Universal Robots PolyScope program: CORAL_QR_l3.urp

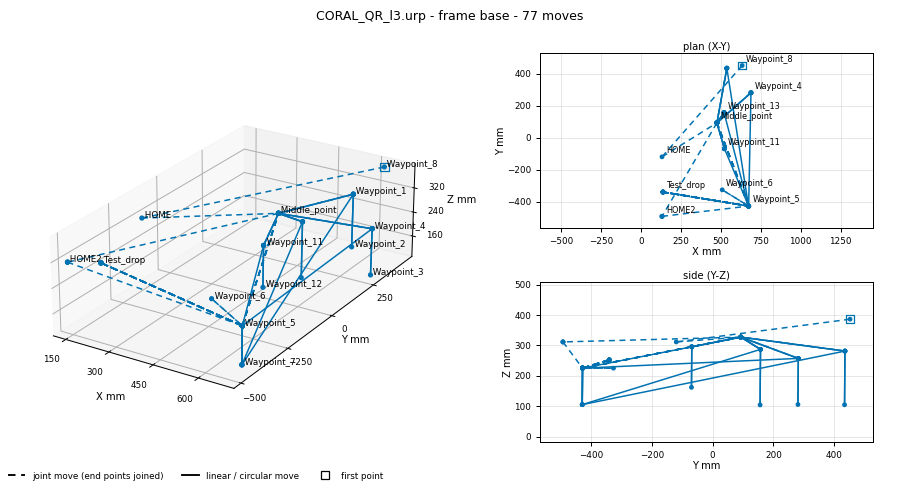
[picture p0: tool path of CORAL_QR_l3.urp in frame base, 77 of 90 moves have a stored position in this frame; points joined in program order, loops and branches not executed]
Program CORAL_QR_l3 (installation=CORAL_installation directory=/programs/usbdisk_0 createdIn=5.13.0 lastSavedIn=5.13.0 robotSerialNumber=20215502618)
Calibrated DH parameters: a=[0.000207, -0.251803, -0.392414, 0.000115, 0.000037, 0]; d=[0.162602, -473.711772, 472.954062, 0.891293, 0.099607, 0.099704]; alpha=[1.571111, -0.000723, 0.005186, 1.570255, -1.569363, 0]; deltaTheta=[0, 0.936857, 5.33632, 0.010013, 0, 0]
InitVariablesNode
Robot Program (runOnlyOnce=false)
  pos_3 := p[0.22031,-0.00393,-0.14981,0.011,-0.001,-1.563]
  pos_4 := p[0.58548,-0.15484,-0.12328,0.011,-0.001,-1.594]
  pos_5 := p[0.38723,-0.17108,-0.15474,0.011,-0.001,-1.594]
  distance := p[0,-0.1,0,0,0,0]
  cont_1 := 1
  cont_2 := 1
  cont_3 := 2
  cont_4 := 2
  cont_5 := 2
  cont_6 := 1
  cont_7 := 1
  no_object := 0
  URCap Gripper Activate (Robotiq_Grippers, Robotiq Inc.) dataModel(ResetAndActivateKey=true)
  URCap External Control (External Control, FZI Research Center for Information Technology)
  MoveL speed 250 mm/s, acceleration 1200 mm/s^2 (useActiveTCP=true) feature=Base
    Waypoint Waypoint_8: TCP in base x=634.227 y=451.95 z=386.422 mm, rx=-1.7963 ry=2.0874 rz=0.1446 rad; joints [201.008, -64.187, 54.919, -99.703, -76.956, 31.795] deg; TCP offset x=0 y=0 z=175.5 mm, rx=0 ry=0 rz=0 rad
  URCap Find Visual Offset (Robotiq_Wrist_Camera, Robotiq Inc.) dataModel(tagModel=[{"_featureName":"CORAL","_automaticMoveEnabled":false,"_ignoreSnapshotPositionEnabled":true,"_skipCloseSnapshotPositionEnabled":false}]); state(isChildrenLocked=true)
    URCap If tag found (Robotiq_Wrist_Camera, Robotiq Inc.)
      URCap Apply Visual Offset (Robotiq_Wrist_Camera, Robotiq Inc.) dataModel(tagModel=[{"_featureName":"CORAL","_appliedEverywhere":false}])
        'Tag found'
        URCap Gripper (Robotiq_Grippers, Robotiq Inc.) dataModel(position=0.0, force=0.0, speed=0.0, positionInDouble=0.0, forceInDouble=0.0, speedInDouble=0.0, slaveIds=[9], blocking=true)
        Loop Forever
          URCap Gripper (Robotiq_Grippers, Robotiq Inc.) dataModel(position=0.0, force=0.0, speed=0.0, positionInDouble=0.0, forceInDouble=0.0, speedInDouble=0.0, slaveIds=[9], blocking=true)
          MoveJ speed 60 deg/s, acceleration 80 deg/s^2 (useActiveTCP=true) feature=Base
            Waypoint HOME: TCP in base x=132.452 y=-119.516 z=311.713 mm, rx=0.0014 ry=-3.1367 rz=0.0022 rad; joints [90.048, -142.3, 117.416, -65.113, -89.996, -0.059] deg
          Wait Condition expression=binary_list_to_integer([digital_in[3],digital_in[4],digital_in[5],digital_in[6],digital_in[7]])==0
          Wait Sleep waitTime=0.25
          Wait Condition expression=binary_list_to_integer([digital_in[3],digital_in[4],digital_in[5],digital_in[6],digital_in[7]])≠0
          Wait Sleep waitTime=0.25
          Script: bit=[digital_in[3],digital_in[4],digital_in[5],digital_in[6],digital_in[7]]
          If binary_list_to_integer(bit)==20
            Wait Condition expression=binary_list_to_integer([digital_in[3],digital_in[4],digital_in[5],digital_in[6],digital_in[7]])==0
            Wait Sleep waitTime=0.25
            Wait Condition expression=binary_list_to_integer([digital_in[3],digital_in[4],digital_in[5],digital_in[6],digital_in[7]])≠0
            Wait Sleep waitTime=0.25
            Script: bit=[digital_in[3],digital_in[4],digital_in[5],digital_in[6],digital_in[7]]
            object := binary_list_to_integer(bit)
            Switch expression=object
              Case (caseValue=11)
                If cont_1≥1
                  MoveJ speed 60 deg/s, acceleration 80 deg/s^2 (useActiveTCP=false) tcp=Robotiq_2F85; feature=Base
                    Waypoint Middle_point: TCP in base x=476.066 y=92.919 z=327.558 mm, rx=-2.1236 ry=2.3147 rz=-0.0001 rad; joints [175.026, -93.413, 90.975, -87.495, -89.706, -0.002] deg
                  MoveL speed 250 mm/s, acceleration 1200 mm/s^2 (useActiveTCP=false) tcp=Robotiq_2F85; feature=CORAL
                    Waypoint Waypoint_1: TCP in base x=538.261 y=435.272 z=281.637 mm, rx=-2.2567 ry=2.1855 rz=-0.0001 rad; joints [207.833, -63.818, 61.827, -87.934, -89.728, 26.021] deg; feature pose in base x=487.974 y=527.462 z=106.955 mm, rx=2.2289 ry=-2.2003 rz=0.002 rad
                    Waypoint Waypoint_2: TCP in base x=537.232 y=433.915 z=104.968 mm, rx=-2.2568 ry=2.1854 rz=-0.0001 rad; joints [207.75, -59.619, 81.826, -112.131, -89.748, 26.056] deg
                    URCap Gripper (Robotiq_Grippers, Robotiq Inc.) dataModel(position=100.0, force=0.0, speed=50.0, positionInDouble=100.0, forceInDouble=0.0, speedInDouble=50.0, slaveIds=[9], blocking=true)
                    Waypoint Waypoint_1: TCP in base x=538.261 y=435.272 z=281.637 mm, rx=-2.2567 ry=2.1855 rz=-0.0001 rad; joints [207.833, -63.818, 61.827, -87.934, -89.728, 26.021] deg
                  cont_1 := cont_1-1
                  no_object := 0
                Else 
                  no_object := 1
                  Popup Message (haltProgram=false message=Out of stock! inputType=Text)
              Case (caseValue=12)
                If cont_2≥1
                  MoveJ speed 60 deg/s, acceleration 80 deg/s^2 (useActiveTCP=false) tcp=Robotiq_2F85; feature=Base
                    Waypoint Middle_point: TCP in base x=476.066 y=92.919 z=327.558 mm, rx=-2.1236 ry=2.3147 rz=-0.0001 rad; joints [175.026, -93.413, 90.975, -87.495, -89.706, -0.002] deg
                  MoveL speed 250 mm/s, acceleration 1200 mm/s^2 (useActiveTCP=false) tcp=Robotiq_2F85; feature=CORAL
                    Waypoint Waypoint_4: TCP in base x=689.362 y=281.81 z=257.546 mm, rx=3.1339 ry=0.0106 rz=-0.0087 rad; joints [192.043, -55.015, 51.59, -86.091, -90.092, -78.333] deg; feature pose in base x=487.974 y=527.462 z=106.955 mm, rx=2.2289 ry=-2.2003 rz=0.002 rad
                    Waypoint Waypoint_3: TCP in base x=688.512 y=280.634 z=105.968 mm, rx=3.1339 ry=0.0105 rz=-0.0087 rad; joints [191.949, -52.35, 69.613, -106.779, -90.102, -78.321] deg
                    URCap Gripper (Robotiq_Grippers, Robotiq Inc.) dataModel(position=100.0, force=0.0, speed=50.0, positionInDouble=100.0, forceInDouble=0.0, speedInDouble=50.0, slaveIds=[9], blocking=true)
                    Waypoint Waypoint_4: TCP in base x=689.362 y=281.81 z=257.546 mm, rx=3.1339 ry=0.0106 rz=-0.0087 rad; joints [192.043, -55.015, 51.59, -86.091, -90.092, -78.333] deg
                  cont_2 := cont_2-1
                  no_object := 0
                Else 
                  no_object := 1
                  Popup Message (haltProgram=false message=Out of stock! inputType=Text)
              Case (caseValue=13)
                If cont_3≥1
                  MoveJ speed 60 deg/s, acceleration 80 deg/s^2 (useActiveTCP=false) tcp=Robotiq_2F85; feature=Base
                    Waypoint Middle_point: TCP in base x=476.066 y=92.919 z=327.558 mm, rx=-2.1236 ry=2.3147 rz=-0.0001 rad; joints [175.026, -93.413, 90.975, -87.495, -89.706, -0.002] deg
                  MoveL speed 250 mm/s, acceleration 1200 mm/s^2 (useActiveTCP=false) tcp=Robotiq_2F85; feature=CORAL
                    Waypoint Variable (Variable): variable=pos_3
                    MoveDirectionNode (selectedDirection=ZPlus toolParams=0.07, 1.2)
                      Until TOOL_CONTACT_DETECTION (allowActions=false retraction=0.02 decelerationAcceleration=3 decelerationAngularAcceleration=34.906585)
                      SuppressedNode
                        Until DISTANCE (allowActions=false deceleration=3 distanceNodeType=STOP) Distance=0.14904; motionParameters(blendRadius=0)
                    URCap Gripper (Robotiq_Grippers, Robotiq Inc.) dataModel(position=100.0, force=0.0, speed=50.0, positionInDouble=100.0, forceInDouble=0.0, speedInDouble=50.0, slaveIds=[9], blocking=true)
                    Waypoint Variable (Variable): variable=pos_3
                    pos_3 := pose_add(pos_3, distance)
                    cont_3 := cont_3-1
                    no_object := 0
                Else 
                  no_object := 1
                  Popup Message (haltProgram=false message=Out of stock! inputType=Text)
              Case (caseValue=14)
                If cont_4≥1
                  MoveJ speed 60 deg/s, acceleration 80 deg/s^2 (useActiveTCP=false) tcp=Robotiq_2F85; feature=Base
                    Waypoint Middle_point: TCP in base x=476.066 y=92.919 z=327.558 mm, rx=-2.1236 ry=2.3147 rz=-0.0001 rad; joints [175.026, -93.413, 90.975, -87.495, -89.706, -0.002] deg
                  MoveL speed 250 mm/s, acceleration 1200 mm/s^2 (useActiveTCP=false) tcp=Robotiq_2F85; feature=CORAL
                    Waypoint Variable (Variable): variable=pos_4
                    MoveDirectionNode (selectedDirection=ZPlus toolParams=0.07, 1.2)
                      Until TOOL_CONTACT_DETECTION (allowActions=false retraction=0.02 decelerationAcceleration=3 decelerationAngularAcceleration=34.906585)
                      SuppressedNode
                        Until DISTANCE (allowActions=false deceleration=3 distanceNodeType=STOP) Distance=0.13; motionParameters(blendRadius=0)
                    URCap Gripper (Robotiq_Grippers, Robotiq Inc.) dataModel(position=100.0, force=0.0, speed=50.0, positionInDouble=100.0, forceInDouble=0.0, speedInDouble=50.0, slaveIds=[9], blocking=true)
                    Waypoint Variable (Variable): variable=pos_4
                    pos_4 := pose_add(pos_4, distance)
                    cont_4 := cont_4-1
                    no_object := 0
                Else 
                  no_object := 1
                  Popup Message (haltProgram=false message=Out of stock! inputType=Text)
              Case (caseValue=15)
                If cont_5≥1
                  MoveJ speed 60 deg/s, acceleration 80 deg/s^2 (useActiveTCP=false) tcp=Robotiq_2F85; feature=Base
                    Waypoint Middle_point: TCP in base x=476.066 y=92.919 z=327.558 mm, rx=-2.1236 ry=2.3147 rz=-0.0001 rad; joints [175.026, -93.413, 90.975, -87.495, -89.706, -0.002] deg
                  MoveL speed 250 mm/s, acceleration 1200 mm/s^2 (useActiveTCP=false) tcp=Robotiq_2F85; feature=CORAL
                    Waypoint Variable (Variable): variable=pos_5
                    MoveDirectionNode (selectedDirection=ZPlus toolParams=0.07, 1.2)
                      Until TOOL_CONTACT_DETECTION (allowActions=false retraction=0.02 decelerationAcceleration=3 decelerationAngularAcceleration=34.906585)
                      SuppressedNode
                        Until DISTANCE (allowActions=false deceleration=3 distanceNodeType=STOP) Distance=0.1485; motionParameters(blendRadius=0)
                    URCap Gripper (Robotiq_Grippers, Robotiq Inc.) dataModel(position=100.0, force=0.0, speed=50.0, positionInDouble=100.0, forceInDouble=0.0, speedInDouble=50.0, slaveIds=[9], blocking=true)
                    Waypoint Variable (Variable): variable=pos_5
                    pos_5 := pose_add(pos_5, distance)
                    cont_5 := cont_5-1
                    no_object := 0
                Else 
                  no_object := 1
                  Popup Message (haltProgram=false message=Out of stock! inputType=Text)
              Case (caseValue=16)
                If cont_6≥1
                  MoveJ speed 60 deg/s, acceleration 80 deg/s^2 (useActiveTCP=false) tcp=Robotiq_2F85; feature=Base
                    Waypoint Middle_point: TCP in base x=476.066 y=92.919 z=327.558 mm, rx=-2.1236 ry=2.3147 rz=-0.0001 rad; joints [175.026, -93.413, 90.975, -87.495, -89.706, -0.002] deg
                  MoveL speed 250 mm/s, acceleration 1200 mm/s^2 (useActiveTCP=false) tcp=Robotiq_2F85; feature=CORAL
                    Waypoint Waypoint_11: TCP in base x=523.11 y=-68.454 z=295.703 mm, rx=3.1197 ry=0.0262 rz=-0.003 rad; joints [158.496, -87.491, 89.855, -92.647, -90.917, -112.404] deg; feature pose in base x=487.974 y=527.462 z=106.955 mm, rx=2.2289 ry=-2.2003 rz=0.002 rad
                    Waypoint Waypoint_12: TCP in base x=522.302 y=-69.494 z=162.29 mm, rx=3.1198 ry=0.0261 rz=-0.0031 rad; joints [158.333, -83.713, 105.789, -112.355, -90.938, -112.468] deg
                    URCap Gripper (Robotiq_Grippers, Robotiq Inc.) dataModel(position=100.0, force=0.0, speed=50.0, positionInDouble=100.0, forceInDouble=0.0, speedInDouble=50.0, slaveIds=[9], blocking=true)
                    Waypoint Waypoint_11: TCP in base x=523.11 y=-68.454 z=295.703 mm, rx=3.1197 ry=0.0262 rz=-0.003 rad; joints [158.496, -87.491, 89.855, -92.647, -90.917, -112.404] deg
                  cont_6 := cont_6-1
                  no_object := 0
                Else 
                  no_object := 1
                  Popup Message (haltProgram=false message=Out of stock! inputType=Text)
              Case (caseValue=17)
                If cont_7≥1
                  MoveJ speed 60 deg/s, acceleration 80 deg/s^2 (useActiveTCP=false) tcp=Robotiq_2F85; feature=Base
                    Waypoint Middle_point: TCP in base x=476.066 y=92.919 z=327.558 mm, rx=-2.1236 ry=2.3147 rz=-0.0001 rad; joints [175.026, -93.413, 90.975, -87.495, -89.706, -0.002] deg
                  MoveL speed 250 mm/s, acceleration 1200 mm/s^2 (useActiveTCP=false) tcp=Robotiq_2F85; feature=CORAL
                    Waypoint Waypoint_13: TCP in base x=520.762 y=157.538 z=287.219 mm, rx=3.1197 ry=0.0264 rz=-0.0033 rad; joints [183.24, -84.793, 88.061, -93.006, -90.961, -87.66] deg; feature pose in base x=487.974 y=527.462 z=106.955 mm, rx=2.2289 ry=-2.2003 rz=0.002 rad
                    Waypoint Waypoint_14: TCP in base x=519.693 y=156.11 z=104.521 mm, rx=3.1197 ry=0.0264 rz=-0.0032 rad; joints [183.068, -77.791, 107.977, -119.927, -91.005, -87.703] deg
                    URCap Gripper (Robotiq_Grippers, Robotiq Inc.) dataModel(position=100.0, force=0.0, speed=50.0, positionInDouble=100.0, forceInDouble=0.0, speedInDouble=50.0, slaveIds=[9], blocking=true)
                    Waypoint Waypoint_13: TCP in base x=520.762 y=157.538 z=287.219 mm, rx=3.1197 ry=0.0264 rz=-0.0033 rad; joints [183.24, -84.793, 88.061, -93.006, -90.961, -87.66] deg
                  cont_7 := cont_7-1
                  no_object := 0
                Else 
                  no_object := 1
                  Popup Message (haltProgram=false message=Out of stock! inputType=Text)
              Case (caseValue=30)
                Popup Message (haltProgram=false message=Action canceled inputType=Text)
                no_object := 1
              Case (caseValue=2147483647)
                no_object := 1
                Popup Message (haltProgram=false message=Incorrect command inputType=Text)
            If no_object==0
              MoveL speed 250 mm/s, acceleration 1200 mm/s^2 (useActiveTCP=true) feature=Base
                Waypoint Middle_point: TCP in base x=476.066 y=92.919 z=327.558 mm, rx=-2.1236 ry=2.3147 rz=-0.0001 rad; joints [175.026, -93.413, 90.975, -87.495, -89.706, -0.002] deg
                SuppressedNode
                  Waypoint Exit_point: TCP in base x=138.592 y=-340.025 z=430.252 mm, rx=-0.0419 ry=-3.1412 rz=0 rad; joints [90.832, -107.12, 86.614, -69.413, -89.733, 2.319] deg
                MoveJ speed 60 deg/s, acceleration 80 deg/s^2 (useActiveTCP=true) feature=Base
                  SuppressedNode
                    Waypoint HOME: TCP in base x=132.452 y=-119.516 z=311.713 mm, rx=0.0014 ry=-3.1367 rz=0.0022 rad; joints [90.048, -142.3, 117.416, -65.113, -89.996, -0.059] deg
                  Waypoint HOME2: TCP in base x=132.456 y=-492.139 z=311.731 mm, rx=0.0014 ry=-3.1367 rz=0.0022 rad; joints [90, -90.004, 90.004, -89.998, -90, 0] deg
                URCap External Control (External Control, FZI Research Center for Information Technology)
                SuppressedNode
                  Waypoint Test_drop: TCP in base x=138.62 y=-340.007 z=252.397 mm, rx=0.0419 ry=3.1413 rz=0 rad; joints [90.789, -110.444, 115.18, -94.656, -89.708, 2.403] deg
              Wait Condition expression=binary_list_to_integer([digital_in[3],digital_in[4],digital_in[5],digital_in[6],digital_in[7]])==0
              Wait Condition expression=binary_list_to_integer([digital_in[3],digital_in[4],digital_in[5],digital_in[6],digital_in[7]])==22
              URCap Gripper (Robotiq_Grippers, Robotiq Inc.) dataModel(position=0.0, force=0.0, speed=50.0, positionInDouble=0.0, forceInDouble=0.0, speedInDouble=50.0, slaveIds=[9], blocking=true)
          ElseIf binary_list_to_integer(bit)==21
            MoveJ speed 60 deg/s, acceleration 80 deg/s^2 (useActiveTCP=false) tcp=Robotiq_2F85; feature=Base
              Waypoint HOME2: TCP in base x=132.456 y=-492.139 z=311.731 mm, rx=0.0014 ry=-3.1367 rz=0.0022 rad; joints [90, -90.004, 90.004, -89.998, -90, 0] deg
            URCap External Control (External Control, FZI Research Center for Information Technology)
            hand_pos := get_actual_tcp_pose()
            sub_option := 50
            Loop While (checkContinuously=false) expression=sub_option==50
              Wait Condition expression=binary_list_to_integer([digital_in[3],digital_in[4],digital_in[5],digital_in[6],digital_in[7]])==0
              Wait Sleep waitTime=0.25
              Wait Condition expression=binary_list_to_integer([digital_in[3],digital_in[4],digital_in[5],digital_in[6],digital_in[7]])≠0
              Wait Sleep waitTime=0.25
              Script: bit=[digital_in[3],digital_in[4],digital_in[5],digital_in[6],digital_in[7]]
              sub_option := binary_list_to_integer(bit)
              If sub_option==22
                URCap Gripper (Robotiq_Grippers, Robotiq Inc.) dataModel(position=100.0, force=0.0, speed=50.0, positionInDouble=100.0, forceInDouble=0.0, speedInDouble=50.0, slaveIds=[9], blocking=true)
                If rq_is_object_detected()== True
                  MoveJ speed 60 deg/s, acceleration 80 deg/s^2 (useActiveTCP=false) tcp=Robotiq_2F85; feature=Base
                    Waypoint HOME2: TCP in base x=132.456 y=-492.139 z=311.731 mm, rx=0.0014 ry=-3.1367 rz=0.0022 rad; joints [90, -90.004, 90.004, -89.998, -90, 0] deg
                  MoveJ speed 60 deg/s, acceleration 80 deg/s^2 (useActiveTCP=false) tcp=Robotiq_2F85; feature=CORAL
                    Waypoint Waypoint_5: TCP in base x=674.764 y=-427.823 z=225.486 mm, rx=0.0319 ry=-3.1243 rz=-0.0059 rad; joints [138.186, -44.607, 38.475, -82.917, -90.23, 47.006] deg; feature pose in base x=487.974 y=527.462 z=106.955 mm, rx=2.2289 ry=-2.2003 rz=0.002 rad
                  MoveL speed 250 mm/s, acceleration 1200 mm/s^2 (useActiveTCP=false) tcp=Robotiq_2F85; feature=CORAL
                    MoveDirectionNode (selectedDirection=ZPlus toolParams=0.07, 1.2)
                      Until TOOL_CONTACT_DETECTION (allowActions=false retraction=NONE decelerationAcceleration=3 decelerationAngularAcceleration=34.906585)
                    URCap Gripper (Robotiq_Grippers, Robotiq Inc.) dataModel(position=0.0, force=0.0, speed=50.0, positionInDouble=0.0, forceInDouble=0.0, speedInDouble=50.0, slaveIds=[9], blocking=true)
                    MoveJ speed 60 deg/s, acceleration 80 deg/s^2 (useActiveTCP=false) tcp=Robotiq_2F85; feature=CORAL
                      Waypoint Waypoint_5: TCP in base x=674.764 y=-427.823 z=225.486 mm, rx=0.0319 ry=-3.1243 rz=-0.0059 rad; joints [138.186, -44.607, 38.475, -82.917, -90.23, 47.006] deg
                      Waypoint Waypoint_6: TCP in base x=509.287 y=-326.093 z=225.43 mm, rx=0.0319 ry=-3.1242 rz=-0.006 rad; joints [134.841, -75.127, 85.478, -99.425, -90.278, 43.766] deg; feature pose in base x=487.974 y=527.462 z=106.955 mm, rx=2.2289 ry=-2.2003 rz=0.002 rad
                    Wait Condition expression=binary_list_to_integer([digital_in[3],digital_in[4],digital_in[5],digital_in[6],digital_in[7]])==0
                    Wait Sleep waitTime=0.25
                    Wait Condition expression=binary_list_to_integer([digital_in[3],digital_in[4],digital_in[5],digital_in[6],digital_in[7]])≠0
                    Wait Sleep waitTime=0.25
                    Script: bit=[digital_in[3],digital_in[4],digital_in[5],digital_in[6],digital_in[7]]
                    object := binary_list_to_integer(bit)
                  Switch expression=object
                    Case (caseValue=1)
                      MoveJ speed 60 deg/s, acceleration 80 deg/s^2 (useActiveTCP=false) tcp=Robotiq_2F85; feature=CORAL
                        Waypoint Waypoint_5: TCP in base x=674.764 y=-427.823 z=225.486 mm, rx=0.0319 ry=-3.1243 rz=-0.0059 rad; joints [138.186, -44.607, 38.475, -82.917, -90.23, 47.006] deg; feature pose in base x=487.974 y=527.462 z=106.955 mm, rx=2.2289 ry=-2.2003 rz=0.002 rad
                      If cont_1==0
                        MoveL speed 250 mm/s, acceleration 1200 mm/s^2 (useActiveTCP=false) tcp=Robotiq_2F85; feature=CORAL
                          SuppressedNode
                            MoveDirectionNode (selectedDirection=ZPlus) feature(featureName=CORAL)
                              Until DISTANCE (allowActions=false deceleration=3 distanceNodeType=STOP) Distance=0.12; motionParameters(blendRadius=0)
                          SuppressedNode
                            Waypoint Waypoint_7: TCP in base x=674.052 y=-428.736 z=105.511 mm, rx=0.0319 ry=-3.1243 rz=-0.0059 rad; joints [138.089, -43.697, 54.45, -99.801, -90.233, 46.995] deg; feature pose in base x=487.974 y=527.462 z=106.955 mm, rx=2.2289 ry=-2.2003 rz=0.002 rad
                          MoveDirectionNode (selectedDirection=ZPlus toolParams=0.07, 1.2)
                            Until TOOL_CONTACT_DETECTION (allowActions=false retraction=0.02 decelerationAcceleration=3 decelerationAngularAcceleration=34.906585)
                          URCap Gripper (Robotiq_Grippers, Robotiq Inc.) dataModel(position=100.0, force=0.0, speed=50.0, positionInDouble=100.0, forceInDouble=0.0, speedInDouble=50.0, slaveIds=[9], blocking=true)
                          Waypoint Waypoint_5: TCP in base x=674.764 y=-427.823 z=225.486 mm, rx=0.0319 ry=-3.1243 rz=-0.0059 rad; joints [138.186, -44.607, 38.475, -82.917, -90.23, 47.006] deg; feature pose in base x=487.974 y=527.462 z=106.955 mm, rx=2.2289 ry=-2.2003 rz=0.002 rad
                          If rq_is_object_detected()== True
                            MoveJ speed 60 deg/s, acceleration 80 deg/s^2 (useActiveTCP=false) tcp=Robotiq_2F85; feature=Base
                              Waypoint Middle_point: TCP in base x=476.066 y=92.919 z=327.558 mm, rx=-2.1236 ry=2.3147 rz=-0.0001 rad; joints [175.026, -93.413, 90.975, -87.495, -89.706, -0.002] deg
                            MoveL speed 250 mm/s, acceleration 1200 mm/s^2 (useActiveTCP=false) tcp=Robotiq_2F85; feature=CORAL
                              Waypoint Waypoint_1: TCP in base x=538.261 y=435.272 z=281.637 mm, rx=-2.2567 ry=2.1855 rz=-0.0001 rad; joints [207.833, -63.818, 61.827, -87.934, -89.728, 26.021] deg; feature pose in base x=487.974 y=527.462 z=106.955 mm, rx=2.2289 ry=-2.2003 rz=0.002 rad
                              MoveDirectionNode (selectedDirection=ZPlus toolParams=0.07, 1.2)
                                Until TOOL_CONTACT_DETECTION (allowActions=false retraction=0 decelerationAcceleration=3 decelerationAngularAcceleration=34.906585)
                              URCap Gripper (Robotiq_Grippers, Robotiq Inc.) dataModel(position=0.0, force=0.0, speed=50.0, positionInDouble=0.0, forceInDouble=0.0, speedInDouble=50.0, slaveIds=[9], blocking=true)
                              Waypoint Waypoint_1: TCP in base x=538.261 y=435.272 z=281.637 mm, rx=-2.2567 ry=2.1855 rz=-0.0001 rad; joints [207.833, -63.818, 61.827, -87.934, -89.728, 26.021] deg
                            cont_1 := cont_1+1
                          Else 
                            Popup Message (haltProgram=false message=Object has been removed, please start again inputType=Text)
                            URCap Gripper (Robotiq_Grippers, Robotiq Inc.) dataModel(position=0.0, force=0.0, speed=50.0, positionInDouble=0.0, forceInDouble=0.0, speedInDouble=50.0, slaveIds=[9], blocking=true)
                      Else 
                        Popup Message (haltProgram=false message=No more space available for this object inputType=Text)
                        MoveL speed 250 mm/s, acceleration 1200 mm/s^2 (useActiveTCP=false) tcp=Robotiq_2F85; feature=CORAL
                          SuppressedNode
                            MoveDirectionNode (selectedDirection=ZPlus) feature(featureName=CORAL)
                              Until DISTANCE (allowActions=false deceleration=3 distanceNodeType=STOP) Distance=0.12; motionParameters(blendRadius=0)
                          Waypoint Waypoint_7: TCP in base x=674.052 y=-428.736 z=105.511 mm, rx=0.0319 ry=-3.1243 rz=-0.0059 rad; joints [138.089, -43.697, 54.45, -99.801, -90.233, 46.995] deg; feature pose in base x=487.974 y=527.462 z=106.955 mm, rx=2.2289 ry=-2.2003 rz=0.002 rad
                        URCap Gripper (Robotiq_Grippers, Robotiq Inc.) dataModel(position=100.0, force=0.0, speed=50.0, positionInDouble=100.0, forceInDouble=0.0, speedInDouble=50.0, slaveIds=[9], blocking=true)
                        MoveL speed 250 mm/s, acceleration 1200 mm/s^2 (useActiveTCP=false) tcp=Robotiq_2F85; feature=CORAL
                          Waypoint Waypoint_5: TCP in base x=674.764 y=-427.823 z=225.486 mm, rx=0.0319 ry=-3.1243 rz=-0.0059 rad; joints [138.186, -44.607, 38.475, -82.917, -90.23, 47.006] deg; feature pose in base x=487.974 y=527.462 z=106.955 mm, rx=2.2289 ry=-2.2003 rz=0.002 rad
                        If rq_is_object_detected()== True
                          MoveJ speed 60 deg/s, acceleration 80 deg/s^2 (useActiveTCP=false) tcp=Robotiq_2F85; feature=Base
                            Waypoint Test_drop: TCP in base x=138.62 y=-340.007 z=252.397 mm, rx=0.0419 ry=3.1413 rz=0 rad; joints [90.789, -110.444, 115.18, -94.656, -89.708, 2.403] deg
                          Wait Condition expression=binary_list_to_integer([digital_in[3],digital_in[4],digital_in[5],digital_in[6],digital_in[7]])==0
                          Wait Condition expression=binary_list_to_integer([digital_in[3],digital_in[4],digital_in[5],digital_in[6],digital_in[7]])==22
                          URCap Gripper (Robotiq_Grippers, Robotiq Inc.) dataModel(position=0.0, force=0.0, speed=50.0, positionInDouble=0.0, forceInDouble=0.0, speedInDouble=50.0, slaveIds=[9], blocking=true)
                        Else 
                          Popup Message (haltProgram=false message=Object has been removed, please start again inputType=Text)
                          URCap Gripper (Robotiq_Grippers, Robotiq Inc.) dataModel(position=0.0, force=0.0, speed=50.0, positionInDouble=0.0, forceInDouble=0.0, speedInDouble=50.0, slaveIds=[9], blocking=true)
                    Case (caseValue=2)
                      MoveJ speed 60 deg/s, acceleration 80 deg/s^2 (useActiveTCP=false) tcp=Robotiq_2F85; feature=CORAL
                        Waypoint Waypoint_5: TCP in base x=674.764 y=-427.823 z=225.486 mm, rx=0.0319 ry=-3.1243 rz=-0.0059 rad; joints [138.186, -44.607, 38.475, -82.917, -90.23, 47.006] deg; feature pose in base x=487.974 y=527.462 z=106.955 mm, rx=2.2289 ry=-2.2003 rz=0.002 rad
                      If cont_2==0
                        MoveL speed 250 mm/s, acceleration 1200 mm/s^2 (useActiveTCP=true) feature=CORAL
                          SuppressedNode
                            MoveDirectionNode (selectedDirection=ZPlus) feature(featureName=CORAL)
                              Until DISTANCE (allowActions=false deceleration=3 distanceNodeType=STOP) Distance=0.115; motionParameters(blendRadius=0)
                          MoveDirectionNode (selectedDirection=ZPlus toolParams=0.07, 1.2)
                            Until TOOL_CONTACT_DETECTION (allowActions=false retraction=0.02 decelerationAcceleration=3 decelerationAngularAcceleration=34.906585)
                          URCap Gripper (Robotiq_Grippers, Robotiq Inc.) dataModel(position=100.0, force=0.0, speed=50.0, positionInDouble=100.0, forceInDouble=0.0, speedInDouble=50.0, slaveIds=[9], blocking=true)
                          Waypoint Waypoint_5: TCP in base x=674.764 y=-427.823 z=225.486 mm, rx=0.0319 ry=-3.1243 rz=-0.0059 rad; joints [138.186, -44.607, 38.475, -82.917, -90.23, 47.006] deg
                          If rq_is_object_detected()== True
                            MoveJ speed 60 deg/s, acceleration 80 deg/s^2 (useActiveTCP=true) feature=Base
                              Waypoint Middle_point: TCP in base x=476.066 y=92.919 z=327.558 mm, rx=-2.1236 ry=2.3147 rz=-0.0001 rad; joints [175.026, -93.413, 90.975, -87.495, -89.706, -0.002] deg
                            MoveL speed 250 mm/s, acceleration 1200 mm/s^2 (useActiveTCP=false) tcp=Robotiq_2F85; feature=CORAL
                              Waypoint Waypoint_4: TCP in base x=689.362 y=281.81 z=257.546 mm, rx=3.1339 ry=0.0106 rz=-0.0087 rad; joints [192.043, -55.015, 51.59, -86.091, -90.092, -78.333] deg; feature pose in base x=487.974 y=527.462 z=106.955 mm, rx=2.2289 ry=-2.2003 rz=0.002 rad
                              MoveDirectionNode (selectedDirection=ZPlus toolParams=0.07, 1.2)
                                Until TOOL_CONTACT_DETECTION (allowActions=false retraction=0 decelerationAcceleration=3 decelerationAngularAcceleration=34.906585)
                              URCap Gripper (Robotiq_Grippers, Robotiq Inc.) dataModel(position=0.0, force=0.0, speed=50.0, positionInDouble=0.0, forceInDouble=0.0, speedInDouble=50.0, slaveIds=[9], blocking=true)
                              Waypoint Waypoint_4: TCP in base x=689.362 y=281.81 z=257.546 mm, rx=3.1339 ry=0.0106 rz=-0.0087 rad; joints [192.043, -55.015, 51.59, -86.091, -90.092, -78.333] deg
                            cont_2 := cont_2+1
                          Else 
                            Popup Message (haltProgram=false message=Object has been removed, please start again inputType=Text)
                            URCap Gripper (Robotiq_Grippers, Robotiq Inc.) dataModel(position=0.0, force=0.0, speed=50.0, positionInDouble=0.0, forceInDouble=0.0, speedInDouble=50.0, slaveIds=[9], blocking=true)
                      Else 
                        Popup Message (haltProgram=false message=No more space available for this object inputType=Text)
                        MoveL speed 250 mm/s, acceleration 1200 mm/s^2 (useActiveTCP=true) feature=CORAL
                          MoveDirectionNode (selectedDirection=ZPlus) feature(featureName=CORAL)
                            Until DISTANCE (allowActions=false deceleration=3 distanceNodeType=STOP) Distance=0.115; motionParameters(blendRadius=0)
                        URCap Gripper (Robotiq_Grippers, Robotiq Inc.) dataModel(position=100.0, force=0.0, speed=50.0, positionInDouble=100.0, forceInDouble=0.0, speedInDouble=50.0, slaveIds=[9], blocking=true)
                        MoveL speed 250 mm/s, acceleration 1200 mm/s^2 (useActiveTCP=false) tcp=Robotiq_2F85; feature=CORAL
                          Waypoint Waypoint_5: TCP in base x=674.764 y=-427.823 z=225.486 mm, rx=0.0319 ry=-3.1243 rz=-0.0059 rad; joints [138.186, -44.607, 38.475, -82.917, -90.23, 47.006] deg; feature pose in base x=487.974 y=527.462 z=106.955 mm, rx=2.2289 ry=-2.2003 rz=0.002 rad
                        If rq_is_object_detected()== True
                          MoveJ speed 60 deg/s, acceleration 80 deg/s^2 (useActiveTCP=true) feature=Base
                            Waypoint Test_drop: TCP in base x=138.62 y=-340.007 z=252.397 mm, rx=0.0419 ry=3.1413 rz=0 rad; joints [90.789, -110.444, 115.18, -94.656, -89.708, 2.403] deg
                          Wait Condition expression=binary_list_to_integer([digital_in[3],digital_in[4],digital_in[5],digital_in[6],digital_in[7]])==0
                          Wait Condition expression=binary_list_to_integer([digital_in[3],digital_in[4],digital_in[5],digital_in[6],digital_in[7]])==22
                          URCap Gripper (Robotiq_Grippers, Robotiq Inc.) dataModel(position=0.0, force=0.0, speed=50.0, positionInDouble=0.0, forceInDouble=0.0, speedInDouble=50.0, slaveIds=[9], blocking=true)
                        Else 
                          Popup Message (haltProgram=false message=Object has been removed, please start again inputType=Text)
                          URCap Gripper (Robotiq_Grippers, Robotiq Inc.) dataModel(position=0.0, force=0.0, speed=50.0, positionInDouble=0.0, forceInDouble=0.0, speedInDouble=50.0, slaveIds=[9], blocking=true)
                    Case (caseValue=3)
                      MoveJ speed 60 deg/s, acceleration 80 deg/s^2 (useActiveTCP=false) tcp=Robotiq_2F85; feature=CORAL
                        Waypoint Waypoint_5: TCP in base x=674.764 y=-427.823 z=225.486 mm, rx=0.0319 ry=-3.1243 rz=-0.0059 rad; joints [138.186, -44.607, 38.475, -82.917, -90.23, 47.006] deg; feature pose in base x=487.974 y=527.462 z=106.955 mm, rx=2.2289 ry=-2.2003 rz=0.002 rad
                      If cont_3<2
                        MoveL speed 250 mm/s, acceleration 1200 mm/s^2 (useActiveTCP=true) feature=CORAL
                          SuppressedNode
                            MoveDirectionNode (selectedDirection=ZPlus) feature(featureName=CORAL)
                              Until DISTANCE (allowActions=false deceleration=3 distanceNodeType=STOP) Distance=0.12; motionParameters(blendRadius=0)
                          SuppressedNode
                            Waypoint Waypoint_7: TCP in base x=674.052 y=-428.736 z=105.511 mm, rx=0.0319 ry=-3.1243 rz=-0.0059 rad; joints [138.089, -43.697, 54.45, -99.801, -90.233, 46.995] deg; feature pose in base x=487.974 y=527.462 z=106.955 mm, rx=2.2289 ry=-2.2003 rz=0.002 rad
                          MoveDirectionNode (selectedDirection=ZPlus toolParams=0.07, 1.2)
                            Until TOOL_CONTACT_DETECTION (allowActions=false retraction=0.02 decelerationAcceleration=3 decelerationAngularAcceleration=34.906585)
                          URCap Gripper (Robotiq_Grippers, Robotiq Inc.) dataModel(position=100.0, force=0.0, speed=50.0, positionInDouble=100.0, forceInDouble=0.0, speedInDouble=50.0, slaveIds=[9], blocking=true)
                          Waypoint Waypoint_5: TCP in base x=674.764 y=-427.823 z=225.486 mm, rx=0.0319 ry=-3.1243 rz=-0.0059 rad; joints [138.186, -44.607, 38.475, -82.917, -90.23, 47.006] deg; feature pose in base x=487.974 y=527.462 z=106.955 mm, rx=2.2289 ry=-2.2003 rz=0.002 rad
                          If rq_is_object_detected()== True
                            MoveJ speed 60 deg/s, acceleration 80 deg/s^2 (useActiveTCP=true) feature=Base
                              Waypoint Middle_point: TCP in base x=476.066 y=92.919 z=327.558 mm, rx=-2.1236 ry=2.3147 rz=-0.0001 rad; joints [175.026, -93.413, 90.975, -87.495, -89.706, -0.002] deg
                            MoveL speed 250 mm/s, acceleration 1200 mm/s^2 (useActiveTCP=true) feature=CORAL
                              pos_3 := pose_sub(pos_3, distance)
                              Waypoint Variable (Variable): variable=pos_3
                              MoveDirectionNode (selectedDirection=ZPlus toolParams=0.07, 1.2)
                                Until TOOL_CONTACT_DETECTION (allowActions=false retraction=0 decelerationAcceleration=3 decelerationAngularAcceleration=34.906585)
                              URCap Gripper (Robotiq_Grippers, Robotiq Inc.) dataModel(position=0.0, force=0.0, speed=50.0, positionInDouble=0.0, forceInDouble=0.0, speedInDouble=50.0, slaveIds=[9], blocking=true)
                              Waypoint Variable (Variable): variable=pos_3
                              cont_3 := cont_3+1
                          Else 
                            Popup Message (haltProgram=false message=Object has been removed, please start again inputType=Text)
                            URCap Gripper (Robotiq_Grippers, Robotiq Inc.) dataModel(position=0.0, force=0.0, speed=50.0, positionInDouble=0.0, forceInDouble=0.0, speedInDouble=50.0, slaveIds=[9], blocking=true)
                      Else 
                        Popup Message (haltProgram=false message=No more space available for this object inputType=Text)
                        MoveL speed 250 mm/s, acceleration 1200 mm/s^2 (useActiveTCP=true) feature=CORAL
                          SuppressedNode
                            MoveDirectionNode (selectedDirection=ZPlus) feature(featureName=CORAL)
                              Until DISTANCE (allowActions=false deceleration=3 distanceNodeType=STOP) Distance=0.12; motionParameters(blendRadius=0)
                          Waypoint Waypoint_7: TCP in base x=674.052 y=-428.736 z=105.511 mm, rx=0.0319 ry=-3.1243 rz=-0.0059 rad; joints [138.089, -43.697, 54.45, -99.801, -90.233, 46.995] deg; feature pose in base x=487.974 y=527.462 z=106.955 mm, rx=2.2289 ry=-2.2003 rz=0.002 rad
                        URCap Gripper (Robotiq_Grippers, Robotiq Inc.) dataModel(position=100.0, force=0.0, speed=50.0, positionInDouble=100.0, forceInDouble=0.0, speedInDouble=50.0, slaveIds=[9], blocking=true)
                        MoveL speed 250 mm/s, acceleration 1200 mm/s^2 (useActiveTCP=false) tcp=Robotiq_2F85; feature=CORAL
                          Waypoint Waypoint_5: TCP in base x=674.764 y=-427.823 z=225.486 mm, rx=0.0319 ry=-3.1243 rz=-0.0059 rad; joints [138.186, -44.607, 38.475, -82.917, -90.23, 47.006] deg; feature pose in base x=487.974 y=527.462 z=106.955 mm, rx=2.2289 ry=-2.2003 rz=0.002 rad
                        If rq_is_object_detected()== True
                          MoveJ speed 60 deg/s, acceleration 80 deg/s^2 (useActiveTCP=true) feature=Base
                            Waypoint Test_drop: TCP in base x=138.62 y=-340.007 z=252.397 mm, rx=0.0419 ry=3.1413 rz=0 rad; joints [90.789, -110.444, 115.18, -94.656, -89.708, 2.403] deg
                          Wait Condition expression=binary_list_to_integer([digital_in[3],digital_in[4],digital_in[5],digital_in[6],digital_in[7]])==0
                          Wait Condition expression=binary_list_to_integer([digital_in[3],digital_in[4],digital_in[5],digital_in[6],digital_in[7]])==22
                          URCap Gripper (Robotiq_Grippers, Robotiq Inc.) dataModel(position=0.0, force=0.0, speed=50.0, positionInDouble=0.0, forceInDouble=0.0, speedInDouble=50.0, slaveIds=[9], blocking=true)
                        Else 
                          Popup Message (haltProgram=false message=Object has been removed, please start again inputType=Text)
                          URCap Gripper (Robotiq_Grippers, Robotiq Inc.) dataModel(position=0.0, force=0.0, speed=50.0, positionInDouble=0.0, forceInDouble=0.0, speedInDouble=50.0, slaveIds=[9], blocking=true)
                    Case (caseValue=4)
                      MoveJ speed 60 deg/s, acceleration 80 deg/s^2 (useActiveTCP=false) tcp=Robotiq_2F85; feature=CORAL
                        Waypoint Waypoint_5: TCP in base x=674.764 y=-427.823 z=225.486 mm, rx=0.0319 ry=-3.1243 rz=-0.0059 rad; joints [138.186, -44.607, 38.475, -82.917, -90.23, 47.006] deg; feature pose in base x=487.974 y=527.462 z=106.955 mm, rx=2.2289 ry=-2.2003 rz=0.002 rad
                      If cont_4<2
                        MoveL speed 250 mm/s, acceleration 1200 mm/s^2 (useActiveTCP=false) tcp=Robotiq_2F85; feature=CORAL
                          SuppressedNode
                            MoveDirectionNode (selectedDirection=ZPlus) feature(featureName=CORAL)
                              Until DISTANCE (allowActions=false deceleration=3 distanceNodeType=STOP) Distance=0.12; motionParameters(blendRadius=0)
                          SuppressedNode
                            Waypoint Waypoint_7: TCP in base x=674.052 y=-428.736 z=105.511 mm, rx=0.0319 ry=-3.1243 rz=-0.0059 rad; joints [138.089, -43.697, 54.45, -99.801, -90.233, 46.995] deg; feature pose in base x=487.974 y=527.462 z=106.955 mm, rx=2.2289 ry=-2.2003 rz=0.002 rad
                          MoveDirectionNode (selectedDirection=ZPlus toolParams=0.07, 1.2)
                            Until TOOL_CONTACT_DETECTION (allowActions=false retraction=0.02 decelerationAcceleration=3 decelerationAngularAcceleration=34.906585)
                          URCap Gripper (Robotiq_Grippers, Robotiq Inc.) dataModel(position=100.0, force=0.0, speed=50.0, positionInDouble=100.0, forceInDouble=0.0, speedInDouble=50.0, slaveIds=[9], blocking=true)
                          Waypoint Waypoint_5: TCP in base x=674.764 y=-427.823 z=225.486 mm, rx=0.0319 ry=-3.1243 rz=-0.0059 rad; joints [138.186, -44.607, 38.475, -82.917, -90.23, 47.006] deg; feature pose in base x=487.974 y=527.462 z=106.955 mm, rx=2.2289 ry=-2.2003 rz=0.002 rad
                          If rq_is_object_detected()== True
                            MoveJ speed 60 deg/s, acceleration 80 deg/s^2 (useActiveTCP=true) feature=Base
                              Waypoint Middle_point: TCP in base x=476.066 y=92.919 z=327.558 mm, rx=-2.1236 ry=2.3147 rz=-0.0001 rad; joints [175.026, -93.413, 90.975, -87.495, -89.706, -0.002] deg
                            MoveL speed 250 mm/s, acceleration 1200 mm/s^2 (useActiveTCP=false) tcp=Robotiq_2F85; feature=CORAL
                              pos_4 := pose_sub(pos_4, distance)
                              Waypoint Variable (Variable): variable=pos_4
                              MoveDirectionNode (selectedDirection=ZPlus toolParams=0.07, 1.2)
                                Until TOOL_CONTACT_DETECTION (allowActions=false retraction=0 decelerationAcceleration=3 decelerationAngularAcceleration=34.906585)
                              URCap Gripper (Robotiq_Grippers, Robotiq Inc.) dataModel(position=0.0, force=0.0, speed=50.0, positionInDouble=0.0, forceInDouble=0.0, speedInDouble=50.0, slaveIds=[9], blocking=true)
                              Waypoint Variable (Variable): variable=pos_4
                              cont_4 := cont_4+1
                          Else 
                            Popup Message (haltProgram=false message=Object has been removed, please start again inputType=Text)
                            URCap Gripper (Robotiq_Grippers, Robotiq Inc.) dataModel(position=0.0, force=0.0, speed=50.0, positionInDouble=0.0, forceInDouble=0.0, speedInDouble=50.0, slaveIds=[9], blocking=true)
                      Else 
                        Popup Message (haltProgram=false message=No more space available for this object inputType=Text)
                        MoveL speed 250 mm/s, acceleration 1200 mm/s^2 (useActiveTCP=false) tcp=Robotiq_2F85; feature=CORAL
                          SuppressedNode
                            MoveDirectionNode (selectedDirection=ZPlus) feature(featureName=CORAL)
                              Until DISTANCE (allowActions=false deceleration=3 distanceNodeType=STOP) Distance=0.12; motionParameters(blendRadius=0)
                          Waypoint Waypoint_7: TCP in base x=674.052 y=-428.736 z=105.511 mm, rx=0.0319 ry=-3.1243 rz=-0.0059 rad; joints [138.089, -43.697, 54.45, -99.801, -90.233, 46.995] deg; feature pose in base x=487.974 y=527.462 z=106.955 mm, rx=2.2289 ry=-2.2003 rz=0.002 rad
                        URCap Gripper (Robotiq_Grippers, Robotiq Inc.) dataModel(position=100.0, force=0.0, speed=50.0, positionInDouble=100.0, forceInDouble=0.0, speedInDouble=50.0, slaveIds=[9], blocking=true)
                        MoveL speed 250 mm/s, acceleration 1200 mm/s^2 (useActiveTCP=false) tcp=Robotiq_2F85; feature=CORAL
                          Waypoint Waypoint_5: TCP in base x=674.764 y=-427.823 z=225.486 mm, rx=0.0319 ry=-3.1243 rz=-0.0059 rad; joints [138.186, -44.607, 38.475, -82.917, -90.23, 47.006] deg; feature pose in base x=487.974 y=527.462 z=106.955 mm, rx=2.2289 ry=-2.2003 rz=0.002 rad
                        If rq_is_object_detected()== True
                          MoveJ speed 60 deg/s, acceleration 80 deg/s^2 (useActiveTCP=true) feature=Base
                            Waypoint Test_drop: TCP in base x=138.62 y=-340.007 z=252.397 mm, rx=0.0419 ry=3.1413 rz=0 rad; joints [90.789, -110.444, 115.18, -94.656, -89.708, 2.403] deg
                          Wait Condition expression=binary_list_to_integer([digital_in[3],digital_in[4],digital_in[5],digital_in[6],digital_in[7]])==0
                          Wait Condition expression=binary_list_to_integer([digital_in[3],digital_in[4],digital_in[5],digital_in[6],digital_in[7]])==22
                          URCap Gripper (Robotiq_Grippers, Robotiq Inc.) dataModel(position=0.0, force=0.0, speed=50.0, positionInDouble=0.0, forceInDouble=0.0, speedInDouble=50.0, slaveIds=[9], blocking=true)
                        Else 
                          Popup Message (haltProgram=false message=Object has been removed, please start again inputType=Text)
                          URCap Gripper (Robotiq_Grippers, Robotiq Inc.) dataModel(position=0.0, force=0.0, speed=50.0, positionInDouble=0.0, forceInDouble=0.0, speedInDouble=50.0, slaveIds=[9], blocking=true)
                    Case (caseValue=5)
                      MoveJ speed 60 deg/s, acceleration 80 deg/s^2 (useActiveTCP=false) tcp=Robotiq_2F85; feature=CORAL
                        Waypoint Waypoint_5: TCP in base x=674.764 y=-427.823 z=225.486 mm, rx=0.0319 ry=-3.1243 rz=-0.0059 rad; joints [138.186, -44.607, 38.475, -82.917, -90.23, 47.006] deg; feature pose in base x=487.974 y=527.462 z=106.955 mm, rx=2.2289 ry=-2.2003 rz=0.002 rad
                      If cont_5<2
                        MoveL speed 250 mm/s, acceleration 1200 mm/s^2 (useActiveTCP=true) feature=CORAL
                          SuppressedNode
                            MoveDirectionNode (selectedDirection=ZPlus) feature(featureName=CORAL)
                              Until DISTANCE (allowActions=false deceleration=3 distanceNodeType=STOP) Distance=0.115; motionParameters(blendRadius=0)
                          MoveDirectionNode (selectedDirection=ZPlus toolParams=0.07, 1.2)
                            Until TOOL_CONTACT_DETECTION (allowActions=false retraction=0.02 decelerationAcceleration=3 decelerationAngularAcceleration=34.906585)
                          URCap Gripper (Robotiq_Grippers, Robotiq Inc.) dataModel(position=100.0, force=0.0, speed=50.0, positionInDouble=100.0, forceInDouble=0.0, speedInDouble=50.0, slaveIds=[9], blocking=true)
                          Waypoint Waypoint_5: TCP in base x=674.764 y=-427.823 z=225.486 mm, rx=0.0319 ry=-3.1243 rz=-0.0059 rad; joints [138.186, -44.607, 38.475, -82.917, -90.23, 47.006] deg
                          If rq_is_object_detected()== True
                            MoveJ speed 60 deg/s, acceleration 80 deg/s^2 (useActiveTCP=true) feature=Base
                              Waypoint Middle_point: TCP in base x=476.066 y=92.919 z=327.558 mm, rx=-2.1236 ry=2.3147 rz=-0.0001 rad; joints [175.026, -93.413, 90.975, -87.495, -89.706, -0.002] deg
                            MoveL speed 250 mm/s, acceleration 1200 mm/s^2 (useActiveTCP=true) feature=CORAL
                              pos_5 := pose_sub(pos_5, distance)
                              Waypoint Variable (Variable): variable=pos_5
                              MoveDirectionNode (selectedDirection=ZPlus toolParams=0.07, 1.2)
                                Until TOOL_CONTACT_DETECTION (allowActions=false retraction=0 decelerationAcceleration=3 decelerationAngularAcceleration=34.906585)
                              URCap Gripper (Robotiq_Grippers, Robotiq Inc.) dataModel(position=0.0, force=0.0, speed=50.0, positionInDouble=0.0, forceInDouble=0.0, speedInDouble=50.0, slaveIds=[9], blocking=true)
                              Waypoint Variable (Variable): variable=pos_5
                              cont_5 := cont_5+1
                          Else 
                            Popup Message (haltProgram=false message=Object has been removed, please start again inputType=Text)
                            URCap Gripper (Robotiq_Grippers, Robotiq Inc.) dataModel(position=0.0, force=0.0, speed=50.0, positionInDouble=0.0, forceInDouble=0.0, speedInDouble=50.0, slaveIds=[9], blocking=true)
                      Else 
                        Popup Message (haltProgram=false message=No more space available for this object inputType=Text)
                        MoveL speed 250 mm/s, acceleration 1200 mm/s^2 (useActiveTCP=true) feature=CORAL
                          MoveDirectionNode (selectedDirection=ZPlus) feature(featureName=CORAL)
                            Until DISTANCE (allowActions=false deceleration=3 distanceNodeType=STOP) Distance=0.115; motionParameters(blendRadius=0)
                        URCap Gripper (Robotiq_Grippers, Robotiq Inc.) dataModel(position=100.0, force=0.0, speed=50.0, positionInDouble=100.0, forceInDouble=0.0, speedInDouble=50.0, slaveIds=[9], blocking=true)
                        MoveL speed 250 mm/s, acceleration 1200 mm/s^2 (useActiveTCP=false) tcp=Robotiq_2F85; feature=CORAL
                          Waypoint Waypoint_5: TCP in base x=674.764 y=-427.823 z=225.486 mm, rx=0.0319 ry=-3.1243 rz=-0.0059 rad; joints [138.186, -44.607, 38.475, -82.917, -90.23, 47.006] deg; feature pose in base x=487.974 y=527.462 z=106.955 mm, rx=2.2289 ry=-2.2003 rz=0.002 rad
                        If rq_is_object_detected()== True
                          MoveJ speed 60 deg/s, acceleration 80 deg/s^2 (useActiveTCP=true) feature=Base
                            Waypoint Test_drop: TCP in base x=138.62 y=-340.007 z=252.397 mm, rx=0.0419 ry=3.1413 rz=0 rad; joints [90.789, -110.444, 115.18, -94.656, -89.708, 2.403] deg
                          Wait Condition expression=binary_list_to_integer([digital_in[3],digital_in[4],digital_in[5],digital_in[6],digital_in[7]])==0
                          Wait Condition expression=binary_list_to_integer([digital_in[3],digital_in[4],digital_in[5],digital_in[6],digital_in[7]])==22
                          URCap Gripper (Robotiq_Grippers, Robotiq Inc.) dataModel(position=0.0, force=0.0, speed=50.0, positionInDouble=0.0, forceInDouble=0.0, speedInDouble=50.0, slaveIds=[9], blocking=true)
                        Else 
                          Popup Message (haltProgram=false message=Object has been removed, please start again inputType=Text)
                          URCap Gripper (Robotiq_Grippers, Robotiq Inc.) dataModel(position=0.0, force=0.0, speed=50.0, positionInDouble=0.0, forceInDouble=0.0, speedInDouble=50.0, slaveIds=[9], blocking=true)
                    Case (caseValue=6)
                      MoveJ speed 60 deg/s, acceleration 80 deg/s^2 (useActiveTCP=false) tcp=Robotiq_2F85; feature=CORAL
                        Waypoint Waypoint_5: TCP in base x=674.764 y=-427.823 z=225.486 mm, rx=0.0319 ry=-3.1243 rz=-0.0059 rad; joints [138.186, -44.607, 38.475, -82.917, -90.23, 47.006] deg; feature pose in base x=487.974 y=527.462 z=106.955 mm, rx=2.2289 ry=-2.2003 rz=0.002 rad
                      If cont_6==0
                        MoveL speed 250 mm/s, acceleration 1200 mm/s^2 (useActiveTCP=false) tcp=Robotiq_2F85; feature=CORAL
                          SuppressedNode
                            MoveDirectionNode (selectedDirection=ZPlus) feature(featureName=CORAL)
                              Until DISTANCE (allowActions=false deceleration=3 distanceNodeType=STOP) Distance=0.071; motionParameters(blendRadius=0)
                          MoveDirectionNode (selectedDirection=ZPlus toolParams=0.07, 1.2)
                            Until TOOL_CONTACT_DETECTION (allowActions=false retraction=0.02 decelerationAcceleration=3 decelerationAngularAcceleration=34.906585)
                          URCap Gripper (Robotiq_Grippers, Robotiq Inc.) dataModel(position=100.0, force=0.0, speed=50.0, positionInDouble=100.0, forceInDouble=0.0, speedInDouble=50.0, slaveIds=[9], blocking=true)
                          Waypoint Waypoint_5: TCP in base x=674.764 y=-427.823 z=225.486 mm, rx=0.0319 ry=-3.1243 rz=-0.0059 rad; joints [138.186, -44.607, 38.475, -82.917, -90.23, 47.006] deg
                          If rq_is_object_detected()== True
                            MoveJ speed 60 deg/s, acceleration 80 deg/s^2 (useActiveTCP=true) feature=Base
                              Waypoint Middle_point: TCP in base x=476.066 y=92.919 z=327.558 mm, rx=-2.1236 ry=2.3147 rz=-0.0001 rad; joints [175.026, -93.413, 90.975, -87.495, -89.706, -0.002] deg
                            MoveL speed 250 mm/s, acceleration 1200 mm/s^2 (useActiveTCP=false) tcp=Robotiq_2F85; feature=CORAL
                              Waypoint Waypoint_11: TCP in base x=523.11 y=-68.454 z=295.703 mm, rx=3.1197 ry=0.0262 rz=-0.003 rad; joints [158.496, -87.491, 89.855, -92.647, -90.917, -112.404] deg; feature pose in base x=487.974 y=527.462 z=106.955 mm, rx=2.2289 ry=-2.2003 rz=0.002 rad
                              MoveDirectionNode (selectedDirection=ZPlus toolParams=0.07, 1.2)
                                Until TOOL_CONTACT_DETECTION (allowActions=false retraction=0 decelerationAcceleration=3 decelerationAngularAcceleration=34.906585)
                              URCap Gripper (Robotiq_Grippers, Robotiq Inc.) dataModel(position=0.0, force=0.0, speed=50.0, positionInDouble=0.0, forceInDouble=0.0, speedInDouble=50.0, slaveIds=[9], blocking=true)
                              Waypoint Waypoint_11: TCP in base x=523.11 y=-68.454 z=295.703 mm, rx=3.1197 ry=0.0262 rz=-0.003 rad; joints [158.496, -87.491, 89.855, -92.647, -90.917, -112.404] deg
                            cont_6 := cont_6+1
                          Else 
                            Popup Message (haltProgram=false message=Object has been removed, please start again inputType=Text)
                            URCap Gripper (Robotiq_Grippers, Robotiq Inc.) dataModel(position=0.0, force=0.0, speed=50.0, positionInDouble=0.0, forceInDouble=0.0, speedInDouble=50.0, slaveIds=[9], blocking=true)
                      Else 
                        Popup Message (haltProgram=false message=No more space available for this object inputType=Text)
                        MoveL speed 250 mm/s, acceleration 1200 mm/s^2 (useActiveTCP=false) tcp=Robotiq_2F85; feature=CORAL
                          MoveDirectionNode (selectedDirection=ZPlus) feature(featureName=CORAL)
                            Until DISTANCE (allowActions=false deceleration=3 distanceNodeType=STOP) Distance=0.071; motionParameters(blendRadius=0)
                        URCap Gripper (Robotiq_Grippers, Robotiq Inc.) dataModel(position=100.0, force=0.0, speed=50.0, positionInDouble=100.0, forceInDouble=0.0, speedInDouble=50.0, slaveIds=[9], blocking=true)
                        MoveL speed 250 mm/s, acceleration 1200 mm/s^2 (useActiveTCP=false) tcp=Robotiq_2F85; feature=CORAL
                          Waypoint Waypoint_5: TCP in base x=674.764 y=-427.823 z=225.486 mm, rx=0.0319 ry=-3.1243 rz=-0.0059 rad; joints [138.186, -44.607, 38.475, -82.917, -90.23, 47.006] deg; feature pose in base x=487.974 y=527.462 z=106.955 mm, rx=2.2289 ry=-2.2003 rz=0.002 rad
                        MoveJ speed 60 deg/s, acceleration 80 deg/s^2 (useActiveTCP=true) feature=Base
                          Waypoint Test_drop: TCP in base x=138.62 y=-340.007 z=252.397 mm, rx=0.0419 ry=3.1413 rz=0 rad; joints [90.789, -110.444, 115.18, -94.656, -89.708, 2.403] deg
                        If rq_is_object_detected()== True
                          Wait Condition expression=binary_list_to_integer([digital_in[3],digital_in[4],digital_in[5],digital_in[6],digital_in[7]])==0
                          Wait Condition expression=binary_list_to_integer([digital_in[3],digital_in[4],digital_in[5],digital_in[6],digital_in[7]])==22
                          URCap Gripper (Robotiq_Grippers, Robotiq Inc.) dataModel(position=0.0, force=0.0, speed=50.0, positionInDouble=0.0, forceInDouble=0.0, speedInDouble=50.0, slaveIds=[9], blocking=true)
                        Else 
                          Popup Message (haltProgram=false message=Object has been removed, please start again inputType=Text)
                          URCap Gripper (Robotiq_Grippers, Robotiq Inc.) dataModel(position=0.0, force=0.0, speed=50.0, positionInDouble=0.0, forceInDouble=0.0, speedInDouble=50.0, slaveIds=[9], blocking=true)
                    Case (caseValue=7)
                      MoveJ speed 60 deg/s, acceleration 80 deg/s^2 (useActiveTCP=false) tcp=Robotiq_2F85; feature=CORAL
                        Waypoint Waypoint_5: TCP in base x=674.764 y=-427.823 z=225.486 mm, rx=0.0319 ry=-3.1243 rz=-0.0059 rad; joints [138.186, -44.607, 38.475, -82.917, -90.23, 47.006] deg; feature pose in base x=487.974 y=527.462 z=106.955 mm, rx=2.2289 ry=-2.2003 rz=0.002 rad
                      If cont_7==0
                        MoveL speed 250 mm/s, acceleration 1200 mm/s^2 (useActiveTCP=false) tcp=Robotiq_2F85; feature=CORAL
                          SuppressedNode
                            MoveDirectionNode (selectedDirection=ZPlus) feature(featureName=CORAL)
                              Until DISTANCE (allowActions=false deceleration=3 distanceNodeType=STOP) Distance=0.12; motionParameters(blendRadius=0)
                          SuppressedNode
                            Waypoint Waypoint_7: TCP in base x=674.052 y=-428.736 z=105.511 mm, rx=0.0319 ry=-3.1243 rz=-0.0059 rad; joints [138.089, -43.697, 54.45, -99.801, -90.233, 46.995] deg; feature pose in base x=487.974 y=527.462 z=106.955 mm, rx=2.2289 ry=-2.2003 rz=0.002 rad
                          MoveDirectionNode (selectedDirection=ZPlus toolParams=0.07, 1.2)
                            Until TOOL_CONTACT_DETECTION (allowActions=false retraction=0.02 decelerationAcceleration=3 decelerationAngularAcceleration=34.906585)
                          URCap Gripper (Robotiq_Grippers, Robotiq Inc.) dataModel(position=100.0, force=0.0, speed=50.0, positionInDouble=100.0, forceInDouble=0.0, speedInDouble=50.0, slaveIds=[9], blocking=true)
                          Waypoint Waypoint_5: TCP in base x=674.764 y=-427.823 z=225.486 mm, rx=0.0319 ry=-3.1243 rz=-0.0059 rad; joints [138.186, -44.607, 38.475, -82.917, -90.23, 47.006] deg; feature pose in base x=487.974 y=527.462 z=106.955 mm, rx=2.2289 ry=-2.2003 rz=0.002 rad
                          If rq_is_object_detected()== True
                            MoveJ speed 60 deg/s, acceleration 80 deg/s^2 (useActiveTCP=true) feature=Base
                              Waypoint Middle_point: TCP in base x=476.066 y=92.919 z=327.558 mm, rx=-2.1236 ry=2.3147 rz=-0.0001 rad; joints [175.026, -93.413, 90.975, -87.495, -89.706, -0.002] deg
                            MoveL speed 250 mm/s, acceleration 1200 mm/s^2 (useActiveTCP=false) tcp=Robotiq_2F85; feature=CORAL
                              Waypoint Waypoint_13: TCP in base x=520.762 y=157.538 z=287.219 mm, rx=3.1197 ry=0.0264 rz=-0.0033 rad; joints [183.24, -84.793, 88.061, -93.006, -90.961, -87.66] deg; feature pose in base x=487.974 y=527.462 z=106.955 mm, rx=2.2289 ry=-2.2003 rz=0.002 rad
                              MoveDirectionNode (selectedDirection=ZPlus toolParams=0.07, 1.2)
                                Until TOOL_CONTACT_DETECTION (allowActions=false retraction=0 decelerationAcceleration=3 decelerationAngularAcceleration=34.906585)
                              URCap Gripper (Robotiq_Grippers, Robotiq Inc.) dataModel(position=0.0, force=0.0, speed=50.0, positionInDouble=0.0, forceInDouble=0.0, speedInDouble=50.0, slaveIds=[9], blocking=true)
                              Waypoint Waypoint_13: TCP in base x=520.762 y=157.538 z=287.219 mm, rx=3.1197 ry=0.0264 rz=-0.0033 rad; joints [183.24, -84.793, 88.061, -93.006, -90.961, -87.66] deg
                            cont_7 := cont_7+1
                          Else 
                            Popup Message (haltProgram=false message=Object has been removed, please start again inputType=Text)
                            URCap Gripper (Robotiq_Grippers, Robotiq Inc.) dataModel(position=0.0, force=0.0, speed=50.0, positionInDouble=0.0, forceInDouble=0.0, speedInDouble=50.0, slaveIds=[9], blocking=true)
                      Else 
                        Popup Message (haltProgram=false message=No more space available for this object inputType=Text)
                        MoveL speed 250 mm/s, acceleration 1200 mm/s^2 (useActiveTCP=false) tcp=Robotiq_2F85; feature=CORAL
                          SuppressedNode
                            MoveDirectionNode (selectedDirection=ZPlus) feature(featureName=CORAL)
                              Until DISTANCE (allowActions=false deceleration=3 distanceNodeType=STOP) Distance=0.12; motionParameters(blendRadius=0)
                          Waypoint Waypoint_7: motionParameters(jointSpeed=1.047198 jointAcceleration=1.396263 cartesianSpeed=0.25 cartesianAcceleration=1.2); TCP in base x=674.052 y=-428.736 z=105.511 mm, rx=0.0319 ry=-3.1243 rz=-0.0059 rad; joints [138.089, -43.697, 54.45, -99.801, -90.233, 46.995] deg
                        URCap Gripper (Robotiq_Grippers, Robotiq Inc.) dataModel(position=100.0, force=0.0, speed=50.0, positionInDouble=100.0, forceInDouble=0.0, speedInDouble=50.0, slaveIds=[9], blocking=true)
                        MoveL speed 250 mm/s, acceleration 1200 mm/s^2 (useActiveTCP=false) tcp=Robotiq_2F85; feature=CORAL
                          Waypoint Waypoint_5: TCP in base x=674.764 y=-427.823 z=225.486 mm, rx=0.0319 ry=-3.1243 rz=-0.0059 rad; joints [138.186, -44.607, 38.475, -82.917, -90.23, 47.006] deg; feature pose in base x=487.974 y=527.462 z=106.955 mm, rx=2.2289 ry=-2.2003 rz=0.002 rad
                        If rq_is_object_detected()== True
                          MoveJ speed 60 deg/s, acceleration 80 deg/s^2 (useActiveTCP=true) feature=Base
                            Waypoint Test_drop: TCP in base x=138.62 y=-340.007 z=252.397 mm, rx=0.0419 ry=3.1413 rz=0 rad; joints [90.789, -110.444, 115.18, -94.656, -89.708, 2.403] deg
                          Wait Condition expression=binary_list_to_integer([digital_in[3],digital_in[4],digital_in[5],digital_in[6],digital_in[7]])==0
                          Wait Condition expression=binary_list_to_integer([digital_in[3],digital_in[4],digital_in[5],digital_in[6],digital_in[7]])==22
                          URCap Gripper (Robotiq_Grippers, Robotiq Inc.) dataModel(position=0.0, force=0.0, speed=50.0, positionInDouble=0.0, forceInDouble=0.0, speedInDouble=50.0, slaveIds=[9], blocking=true)
                        Else 
                          Popup Message (haltProgram=false message=Object has been removed, please start again inputType=Text)
                    Case (caseValue=8)
                      Popup Message (haltProgram=false message=Object not identified inputType=Text)
                      MoveJ speed 60 deg/s, acceleration 80 deg/s^2 (useActiveTCP=false) tcp=Robotiq_2F85; feature=CORAL
                        Waypoint Waypoint_5: TCP in base x=674.764 y=-427.823 z=225.486 mm, rx=0.0319 ry=-3.1243 rz=-0.0059 rad; joints [138.186, -44.607, 38.475, -82.917, -90.23, 47.006] deg; feature pose in base x=487.974 y=527.462 z=106.955 mm, rx=2.2289 ry=-2.2003 rz=0.002 rad
                      MoveL speed 70 mm/s, acceleration 1200 mm/s^2 (useActiveTCP=false) tcp=Robotiq_2F85; feature=CORAL
                        MoveDirectionNode (selectedDirection=ZPlus)
                          Until TOOL_CONTACT_DETECTION (allowActions=false retraction=0.02 decelerationAcceleration=3 decelerationAngularAcceleration=34.906585)
                        URCap Gripper (Robotiq_Grippers, Robotiq Inc.) dataModel(position=100.0, force=0.0, speed=50.0, positionInDouble=100.0, forceInDouble=0.0, speedInDouble=50.0, slaveIds=[9], blocking=true)
                        Waypoint Waypoint_5: TCP in base x=674.764 y=-427.823 z=225.486 mm, rx=0.0319 ry=-3.1243 rz=-0.0059 rad; joints [138.186, -44.607, 38.475, -82.917, -90.23, 47.006] deg
                        If rq_is_object_detected()== True
                          MoveJ speed 60 deg/s, acceleration 80 deg/s^2 (useActiveTCP=true) feature=Base
                            SuppressedNode
                              Waypoint Test_drop: TCP in base x=138.62 y=-340.007 z=252.397 mm, rx=0.0419 ry=3.1413 rz=0 rad; joints [90.789, -110.444, 115.18, -94.656, -89.708, 2.403] deg
                            Waypoint Variable (Variable): variable=hand_pos
                          Wait Condition expression=binary_list_to_integer([digital_in[3],digital_in[4],digital_in[5],digital_in[6],digital_in[7]])==0
                          Wait Condition expression=binary_list_to_integer([digital_in[3],digital_in[4],digital_in[5],digital_in[6],digital_in[7]])==22
                          URCap Gripper (Robotiq_Grippers, Robotiq Inc.) dataModel(position=0.0, force=0.0, speed=50.0, positionInDouble=0.0, forceInDouble=0.0, speedInDouble=50.0, slaveIds=[9], blocking=true)
                        Else 
                          Popup Message (haltProgram=false message=Object has been removed, please start again inputType=Text)
                          URCap Gripper (Robotiq_Grippers, Robotiq Inc.) dataModel(position=0.0, force=0.0, speed=50.0, positionInDouble=0.0, forceInDouble=0.0, speedInDouble=50.0, slaveIds=[9], blocking=true)
                    Case (caseValue=30)
                      Popup Message (haltProgram=false message=Action canceled inputType=Text)
                    Case (caseValue=2147483647)
                      Popup Message (haltProgram=false message=Incorrect command inputType=Text)
                Else 
                  Popup Message (haltProgram=false message=Object not grabbed, please approach the object to the gripper again inputType=Text)
                  sub_option := 50
                  URCap Gripper (Robotiq_Grippers, Robotiq Inc.) dataModel(position=0.0, force=0.0, speed=0.0, positionInDouble=0.0, forceInDouble=0.0, speedInDouble=0.0, slaveIds=[9], blocking=true)
              ElseIf sub_option==30
                Popup Message (haltProgram=false message=Action canceled inputType=Text)
                sub_option := 100
              Else 
                Popup Message (haltProgram=false message=Invalid action, please try again inputType=Text)
                sub_option := 50
          Else 
            Popup Message (haltProgram=false message=Invalid action, please try again inputType=Text)
    URCap If tag not found (Robotiq_Wrist_Camera, Robotiq Inc.)
      'Missing tag'
      Popup Message (haltProgram=false message=Tag not found! inputType=Text)
      Halt
